{attribute 'GeneratedUsingTerminal: EL3314-0000-0016'}
{attribute addProperty BoxType "EL3314-0000-0016"}
{attribute addProperty Id "TC_Inputs_Channel_1AT %I*TC_Inputs_Channel_EA9DF21E9TC_Inputs_Channel_2AT %I*TC_Inputs_Channel_EA9DF21E9TC_Inputs_Channel_3AT %I*TC_Inputs_Channel_EA9DF21E9TC_Inputs_Channel_4AT %I*TC_Inputs_Channel_EA9DF21E9WcStateAT %I*WcState_9091E0EB2InfoDataAT %I*InfoData_94A18F5E2"}
{attribute addProperty CRC "3640132412"}
{attribute addProperty Size "40"}
TYPE EL3314_D8F8033C EXTENDS EtcSlaveTerminalBase_947E5A46 :
STRUCT
	{attribute addProperty Name "TC_Inputs_Channel_1"}
	TC_Inputs_Channel_1 : TC_Inputs_Channel_EA9DF21E;
	{attribute addProperty Name "TC_Inputs_Channel_2"}
	TC_Inputs_Channel_2 : TC_Inputs_Channel_EA9DF21E;
	{attribute addProperty Name "TC_Inputs_Channel_3"}
	TC_Inputs_Channel_3 : TC_Inputs_Channel_EA9DF21E;
	{attribute addProperty Name "TC_Inputs_Channel_4"}
	TC_Inputs_Channel_4 : TC_Inputs_Channel_EA9DF21E;
	{attribute addProperty Name "WcState"}
	WcState : WcState_9091E0EB;
	{attribute addProperty Name "InfoData"}
	InfoData : InfoData_94A18F5E;
END_STRUCT
END_TYPE

(* stored: Version 1.2.0.0, ProductVersion 3.1.4024.9
   DUT EL3314_D8F8033C: Id {0c24e5dc-0462-4f9b-a8cd-f40dc10f6ae1} *)
